// TIA Portal V20 program export: 0 tag tables, 0 data types, 2 data blocks, 3 code blocks (in call order from the OBs), 0 instance data blocks

DATA_BLOCK "DB_Alarmas"   // DB3
{ S7_Optimized_Access := 'TRUE' }
// stored: MemoryReserve 100
   VAR
      Registro_Fallos : Word;
   END_VAR
BEGIN
END_DATA_BLOCK

DATA_BLOCK "DB_Manual"   // DB4
{ S7_Optimized_Access := 'TRUE' }
// stored: MemoryReserve 100
   VAR
      Modo_Activo : Bool;
      HMI_C1_Sale : Bool;
      HMI_C1_Entra : Bool;
      HMI_C2_Sale : Bool;
      HMI_C2_Entra : Bool;
      "HMI_M_90°" : Bool;
      "HMI_M_0°" : Bool;
   END_VAR
BEGIN
END_DATA_BLOCK

ORGANIZATION_BLOCK "Main"   // OB1, LAD, ProgramCycle
TITLE = "Main Program Sweep (Cycle)"
{ S7_Optimized_Access := 'TRUE' }
// stored: SetENOAutomatically false
   VAR_INPUT
      Initial_Call : Bool;   // Initial call of this OB
      Remanence : Bool;   // =True, if remanent data are available
   END_VAR
BEGIN

REGION Network 1
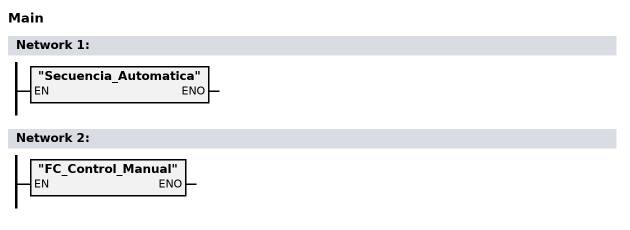
   RUNG wire#powerrail
      "Secuencia_Automatica"()
   END_RUNG
   // the same network as SCL:
   "Secuencia_Automatica"();
END_REGION

REGION Network 2
   RUNG wire#powerrail
      "FC_Control_Manual"()
   END_RUNG
   // the same network as SCL:
   "FC_Control_Manual"();
END_REGION
END_ORGANIZATION_BLOCK

FUNCTION "Secuencia_Automatica" : Void   // FC1, LAD
{ S7_Optimized_Access := 'TRUE' }
// stored: SetENOAutomatically false
BEGIN

REGION Network 1: Relé maestro de ciclo continuo (Autorretención de START)
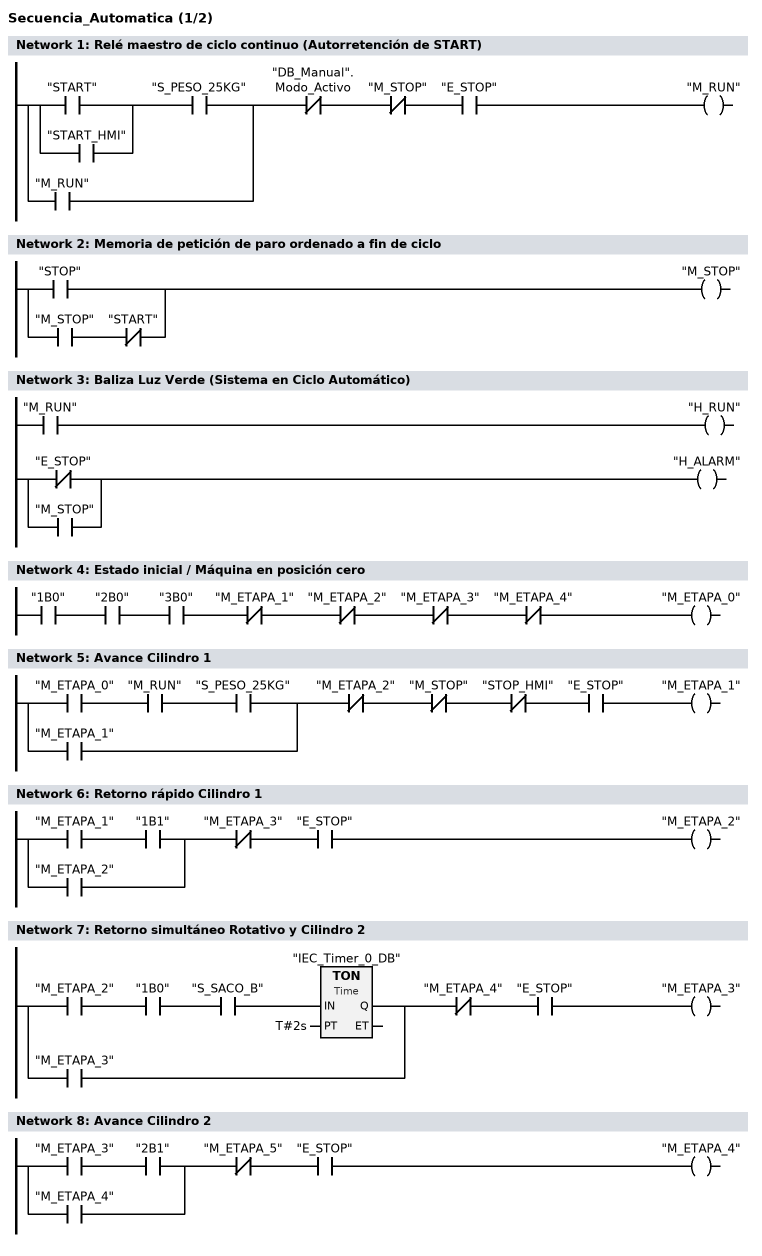
   RUNG wire#powerrail
      Contact( "START" )
      wire#w1
      Contact( "S_PESO_25KG" )
      wire#w2
      I_Contact( "DB_Manual".Modo_Activo )
      I_Contact( "M_STOP" )
      Contact( "E_STOP" )
      Coil( "M_RUN" )
   END_RUNG
   RUNG wire#powerrail
      Contact( "START_HMI" )
   END_RUNG wire#w1
   RUNG wire#powerrail
      Contact( "M_RUN" )
   END_RUNG wire#w2
   // the same network as SCL:
   "M_RUN" := ((("START" OR "START_HMI") AND "S_PESO_25KG") OR "M_RUN") AND NOT "DB_Manual".Modo_Activo AND NOT "M_STOP" AND "E_STOP";
END_REGION

REGION Network 2: Memoria de petición de paro ordenado a fin de ciclo
   RUNG wire#powerrail
      Contact( "STOP" )
      wire#w1
      Coil( "M_STOP" )
   END_RUNG
   RUNG wire#powerrail
      Contact( "M_STOP" )
      I_Contact( "START" )
   END_RUNG wire#w1
   // the same network as SCL:
   "M_STOP" := "STOP" OR ("M_STOP" AND NOT "START");
END_REGION

REGION Network 3: Baliza Luz Verde (Sistema en Ciclo Automático)
   RUNG wire#powerrail
      Contact( "M_RUN" )
      Coil( "H_RUN" )
   END_RUNG
   RUNG wire#powerrail
      I_Contact( "E_STOP" )
      wire#w1
      Coil( "H_ALARM" )
   END_RUNG
   RUNG wire#powerrail
      Contact( "M_STOP" )
   END_RUNG wire#w1
   // the same network as SCL:
   "H_RUN" := "M_RUN";
   "H_ALARM" := NOT "E_STOP" OR "M_STOP";
END_REGION

REGION Network 4: Estado inicial / Máquina en posición cero
   RUNG wire#powerrail
      Contact( "1B0" )
      Contact( "2B0" )
      Contact( "3B0" )
      I_Contact( "M_ETAPA_1" )
      I_Contact( "M_ETAPA_2" )
      I_Contact( "M_ETAPA_3" )
      I_Contact( "M_ETAPA_4" )
      Coil( "M_ETAPA_0" )
   END_RUNG
   // the same network as SCL:
   "M_ETAPA_0" := "1B0" AND "2B0" AND "3B0" AND NOT "M_ETAPA_1" AND NOT "M_ETAPA_2" AND NOT "M_ETAPA_3" AND NOT "M_ETAPA_4";
END_REGION

REGION Network 5: Avance Cilindro 1
   RUNG wire#powerrail
      Contact( "M_ETAPA_0" )
      Contact( "M_RUN" )
      Contact( "S_PESO_25KG" )
      wire#w1
      I_Contact( "M_ETAPA_2" )
      I_Contact( "M_STOP" )
      I_Contact( "STOP_HMI" )
      Contact( "E_STOP" )
      Coil( "M_ETAPA_1" )
   END_RUNG
   RUNG wire#powerrail
      Contact( "M_ETAPA_1" )
   END_RUNG wire#w1
   // the same network as SCL:
   "M_ETAPA_1" := (("M_ETAPA_0" AND "M_RUN" AND "S_PESO_25KG") OR "M_ETAPA_1") AND NOT "M_ETAPA_2" AND NOT "M_STOP" AND NOT "STOP_HMI" AND "E_STOP";
END_REGION

REGION Network 6: Retorno rápido Cilindro 1
   RUNG wire#powerrail
      Contact( "M_ETAPA_1" )
      Contact( "1B1" )
      wire#w1
      I_Contact( "M_ETAPA_3" )
      Contact( "E_STOP" )
      Coil( "M_ETAPA_2" )
   END_RUNG
   RUNG wire#powerrail
      Contact( "M_ETAPA_2" )
   END_RUNG wire#w1
   // the same network as SCL:
   "M_ETAPA_2" := (("M_ETAPA_1" AND "1B1") OR "M_ETAPA_2") AND NOT "M_ETAPA_3" AND "E_STOP";
END_REGION

REGION Network 7: Retorno simultáneo Rotativo y Cilindro 2
   RUNG wire#powerrail
      Contact( "M_ETAPA_2" )
      Contact( "1B0" )
      Contact( "S_SACO_B" )
      { S7_Templates := "time_type := Time" } "IEC_Timer_0_DB".TON(pt := T#2s, et =>)
      wire#w1
      I_Contact( "M_ETAPA_4" )
      Contact( "E_STOP" )
      Coil( "M_ETAPA_3" )
   END_RUNG
   RUNG wire#powerrail
      Contact( "M_ETAPA_3" )
   END_RUNG wire#w1
   // the same network as SCL:
   "IEC_Timer_0_DB".TON(IN := "M_ETAPA_2" AND "1B0" AND "S_SACO_B", PT := T#2s);
   "M_ETAPA_3" := ("IEC_Timer_0_DB".Q OR "M_ETAPA_3") AND NOT "M_ETAPA_4" AND "E_STOP";
END_REGION

REGION Network 8: Avance Cilindro 2
   RUNG wire#powerrail
      Contact( "M_ETAPA_3" )
      Contact( "2B1" )
      wire#w1
      I_Contact( "M_ETAPA_5" )
      Contact( "E_STOP" )
      Coil( "M_ETAPA_4" )
   END_RUNG
   RUNG wire#powerrail
      Contact( "M_ETAPA_4" )
   END_RUNG wire#w1
   // the same network as SCL:
   "M_ETAPA_4" := (("M_ETAPA_3" AND "2B1") OR "M_ETAPA_4") AND NOT "M_ETAPA_5" AND "E_STOP";
END_REGION

REGION Network 9: Retorno simultáneo Rotativo y Cilindro 2
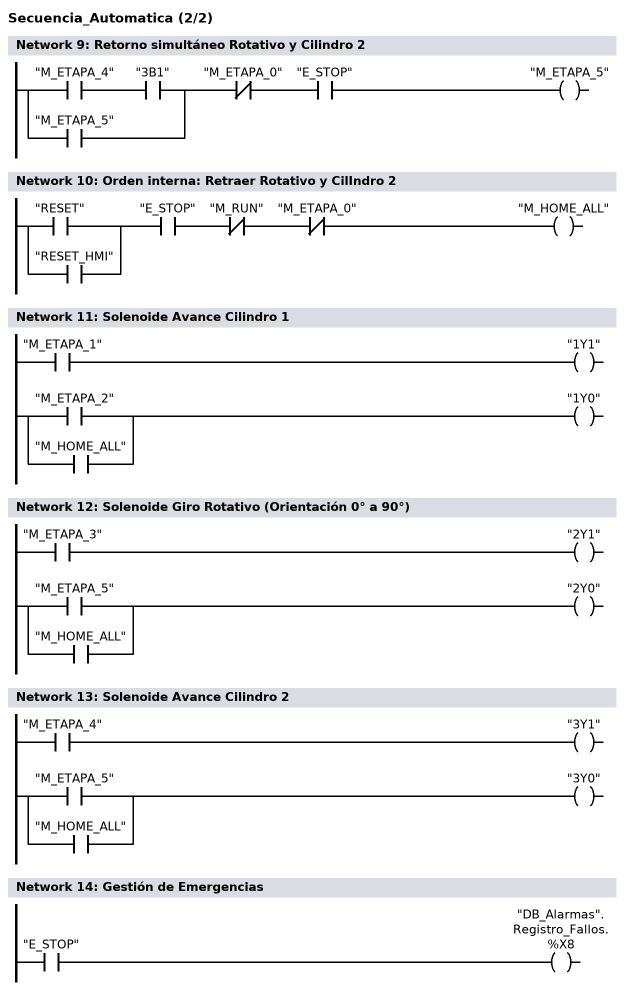
   RUNG wire#powerrail
      Contact( "M_ETAPA_4" )
      Contact( "3B1" )
      wire#w1
      I_Contact( "M_ETAPA_0" )
      Contact( "E_STOP" )
      Coil( "M_ETAPA_5" )
   END_RUNG
   RUNG wire#powerrail
      Contact( "M_ETAPA_5" )
   END_RUNG wire#w1
   // the same network as SCL:
   "M_ETAPA_5" := (("M_ETAPA_4" AND "3B1") OR "M_ETAPA_5") AND NOT "M_ETAPA_0" AND "E_STOP";
END_REGION

REGION Network 10: Orden interna: Retraer Rotativo y CilIndro 2
   RUNG wire#powerrail
      Contact( "RESET" )
      wire#w1
      Contact( "E_STOP" )
      I_Contact( "M_RUN" )
      I_Contact( "M_ETAPA_0" )
      Coil( "M_HOME_ALL" )
   END_RUNG
   RUNG wire#powerrail
      Contact( "RESET_HMI" )
   END_RUNG wire#w1
   // the same network as SCL:
   "M_HOME_ALL" := ("RESET" OR "RESET_HMI") AND "E_STOP" AND NOT "M_RUN" AND NOT "M_ETAPA_0";
END_REGION

REGION Network 11: Solenoide Avance Cilindro 1
   RUNG wire#powerrail
      Contact( "M_ETAPA_1" )
      Coil( "1Y1" )
   END_RUNG
   RUNG wire#powerrail
      Contact( "M_ETAPA_2" )
      wire#w1
      Coil( "1Y0" )
   END_RUNG
   RUNG wire#powerrail
      Contact( "M_HOME_ALL" )
   END_RUNG wire#w1
   // the same network as SCL:
   "1Y1" := "M_ETAPA_1";
   "1Y0" := "M_ETAPA_2" OR "M_HOME_ALL";
END_REGION

REGION Network 12: Solenoide Giro Rotativo (Orientación 0° a 90°)
   RUNG wire#powerrail
      Contact( "M_ETAPA_3" )
      Coil( "2Y1" )
   END_RUNG
   RUNG wire#powerrail
      Contact( "M_ETAPA_5" )
      wire#w1
      Coil( "2Y0" )
   END_RUNG
   RUNG wire#powerrail
      Contact( "M_HOME_ALL" )
   END_RUNG wire#w1
   // the same network as SCL:
   "2Y1" := "M_ETAPA_3";
   "2Y0" := "M_ETAPA_5" OR "M_HOME_ALL";
END_REGION

REGION Network 13: Solenoide Avance Cilindro 2
   RUNG wire#powerrail
      Contact( "M_ETAPA_4" )
      Coil( "3Y1" )
   END_RUNG
   RUNG wire#powerrail
      Contact( "M_ETAPA_5" )
      wire#w1
      Coil( "3Y0" )
   END_RUNG
   RUNG wire#powerrail
      Contact( "M_HOME_ALL" )
   END_RUNG wire#w1
   // the same network as SCL:
   "3Y1" := "M_ETAPA_4";
   "3Y0" := "M_ETAPA_5" OR "M_HOME_ALL";
END_REGION

REGION Network 14: Gestión de Emergencias
   RUNG wire#powerrail
      Contact( "E_STOP" )
      Coil( "DB_Alarmas".Registro_Fallos.%X8 )
   END_RUNG
   // the same network as SCL:
   "DB_Alarmas".Registro_Fallos.%X8 := "E_STOP";
END_REGION
END_FUNCTION

FUNCTION "FC_Control_Manual" : Void   // FC2, LAD
{ S7_Optimized_Access := 'TRUE' }
// stored: SetENOAutomatically false
BEGIN

REGION Network 1: Solenoide Salida Cilindro 1
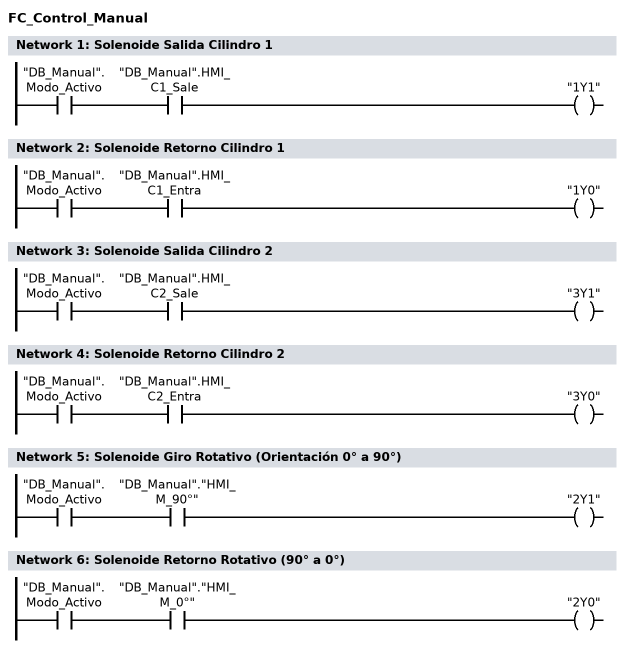
   RUNG wire#powerrail
      Contact( "DB_Manual".Modo_Activo )
      Contact( "DB_Manual".HMI_C1_Sale )
      Coil( "1Y1" )
   END_RUNG
   // the same network as SCL:
   "1Y1" := "DB_Manual".Modo_Activo AND "DB_Manual".HMI_C1_Sale;
END_REGION

REGION Network 2: Solenoide Retorno Cilindro 1
   RUNG wire#powerrail
      Contact( "DB_Manual".Modo_Activo )
      Contact( "DB_Manual".HMI_C1_Entra )
      Coil( "1Y0" )
   END_RUNG
   // the same network as SCL:
   "1Y0" := "DB_Manual".Modo_Activo AND "DB_Manual".HMI_C1_Entra;
END_REGION

REGION Network 3: Solenoide Salida Cilindro 2
   RUNG wire#powerrail
      Contact( "DB_Manual".Modo_Activo )
      Contact( "DB_Manual".HMI_C2_Sale )
      Coil( "3Y1" )
   END_RUNG
   // the same network as SCL:
   "3Y1" := "DB_Manual".Modo_Activo AND "DB_Manual".HMI_C2_Sale;
END_REGION

REGION Network 4: Solenoide Retorno Cilindro 2
   RUNG wire#powerrail
      Contact( "DB_Manual".Modo_Activo )
      Contact( "DB_Manual".HMI_C2_Entra )
      Coil( "3Y0" )
   END_RUNG
   // the same network as SCL:
   "3Y0" := "DB_Manual".Modo_Activo AND "DB_Manual".HMI_C2_Entra;
END_REGION

REGION Network 5: Solenoide Giro Rotativo (Orientación 0° a 90°)
   RUNG wire#powerrail
      Contact( "DB_Manual".Modo_Activo )
      Contact( "DB_Manual"."HMI_M_90°" )
      Coil( "2Y1" )
   END_RUNG
   // the same network as SCL:
   "2Y1" := "DB_Manual".Modo_Activo AND "DB_Manual"."HMI_M_90°";
END_REGION

REGION Network 6: Solenoide Retorno Rotativo (90° a 0°)
   RUNG wire#powerrail
      Contact( "DB_Manual".Modo_Activo )
      Contact( "DB_Manual"."HMI_M_0°" )
      Coil( "2Y0" )
   END_RUNG
   // the same network as SCL:
   "2Y0" := "DB_Manual".Modo_Activo AND "DB_Manual"."HMI_M_0°";
END_REGION
END_FUNCTION
